FUNCTION_BLOCK CAT_Robotino_HMI (* Service Interface Function Block Type *)
  (* Standard: 61499-2 *)
  (* Version 0.0, 26/10/2022, Pranay Jhunjhunwala, Schneider Electric, template *)
  PACKAGE Main;
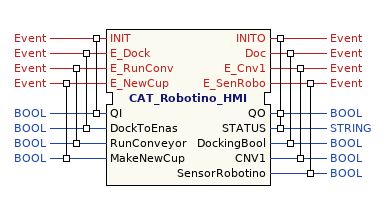
  EVENT_INPUT
    INIT WITH QI;
    E_Dock WITH DockToEnas;
    E_RunConv WITH RunConveyor;
    E_NewCup WITH MakeNewCup;
  END_EVENT
  EVENT_OUTPUT
    INITO WITH QO, STATUS;
    Doc WITH DockingBool;
    E_Cnv1 WITH CNV1;
    E_SenRobo WITH SensorRobotino;
  END_EVENT
  VAR_INPUT
    QI : BOOL;
    DockToEnas : BOOL;
    RunConveyor : BOOL;
    MakeNewCup : BOOL;
  END_VAR
  VAR_OUTPUT
    QO : BOOL; (* Event Output Qualifier *)
    STATUS : STRING; (* Service Status *)
    DockingBool : BOOL;
    CNV1 : BOOL;
    SensorRobotino : BOOL;
  END_VAR
  SERVICE /
    SEQUENCE 
    END_SEQUENCE
  END_SERVICE
END_FUNCTION_BLOCK
